PROGRAM ManualHorAxis
VAR
END_VAR

HAVL.axis.ReadStatus();

IF HAVL.extend AND NOT(HAVL.endStop) THEN
	HAVL.lastExtend := TRUE;
	HAVL.lastRetract := FALSE;
END_IF

IF HAVL.retract AND NOT(HAVL.endStop) THEN
	HAVL.lastExtend := FALSE;
	HAVL.lastRetract := TRUE;
END_IF

HAVL.axisPower(
	Axis:= HAVL.axis,
	Enable:= HAVL.enable,
	Enable_Positive:= HAVL.enable,
	Enable_Negative:= HAVL.enable,
	Override:= HAVL.override,
	BufferMode:= ,
	Options:= ,
	Status=> HAVL.running,
	Busy=> ,
	Active=> ,
	Error=> ,
	ErrorID=> HAVL.currentError
);

HAVL.axisMoveManual(
	Axis:= HAVL.axis,
	JogForward:= (HAVL.extend AND (NOT(HAVL.endStop) OR (HAVL.endStop AND HAVL.lastRetract))),
	JogBackwards:= (HAVL.retract AND (NOT(HAVL.endStop) OR (HAVL.endStop AND HAVL.lastExtend))),
	Mode:= ,
	Position:= ,
	Velocity:= ,
	Acceleration:= ,
	Deceleration:= ,
	Jerk:= ,
	Done=> HAVL.done,
	Busy=> HAVL.busy,
	Active=> ,
	CommandAborted=> ,
	Error=> ,
	ErrorID=> HAVL.currentError
);
	
IF HAVL.busy THEN
	HAVL.axisReadActualPosition(Axis := HAVL.axis, Enable := TRUE, Valid=>, Busy=>, Error=>, ErrorID=>, Position=> HAVL.actualPosition);
END_IF
HAVL.actualPositionInt := LREAL_TO_INT(HAVL.actualPosition);

HAVL.axisErrorReset(Axis := HAVL.axis, Execute := HAVL.resetError, Done =>, Error =>, ErrorID => HAVL.currentError);

END_PROGRAM

(* stored: Version 1.1.0.1, ProductVersion 3.1.4024.6
   POU ManualHorAxis: Id {880819fa-648e-4916-b2f4-018c51c85792}, SpecialFunc None *)
